INTERFACE I_Reflection

{attribute 'OPC.UA.DA.Property' := '1'}
{attribute 'monitoring' := 'call'}
PROPERTY PUBLIC P_Class : STRING(255)
GET
END_GET
END_PROPERTY

{attribute 'OPC.UA.DA.Property' := '1'}
{attribute 'monitoring' := 'call'}
PROPERTY PUBLIC P_Comment : STRING(255)
GET
END_GET
END_PROPERTY

{attribute 'OPC.UA.DA.Property' := '1'}
{attribute 'monitoring' := 'call'}
PROPERTY PUBLIC P_ID : STRING(25)
GET
END_GET
SET
END_SET
END_PROPERTY

{attribute 'OPC.UA.DA.Property' := '1'}
{attribute 'monitoring' := 'call'}
PROPERTY PUBLIC P_Instance : STRING(255)
GET
END_GET
END_PROPERTY

{attribute 'OPC.UA.DA.Property' := '1'}
{attribute 'monitoring' := 'call'}
PROPERTY PUBLIC P_Timestamp : DT
GET
END_GET
END_PROPERTY

END_INTERFACE

(* stored: Version 1.1.0.1
   Itf I_Reflection: Id {62aeab96-2429-49a4-b102-a608a3391a9f}
   Property P_Class: Id {cbc4d901-48b2-4e97-9d77-884fb0854f2f}
   Get Get: Id {9ab4d9fd-c087-473a-be35-5661f24836f2}
   Property P_Comment: Id {f8cad2c1-c823-4908-b22c-bf669c46c6ef}
   Get Get: Id {83892f6a-bbdf-4950-9818-7b29a5f63cc7}
   Property P_ID: Id {1189c098-5eec-0d68-18e7-7614f6e3884e}
   Get Get: Id {119ce5e0-3bc0-09ab-2641-05ccee762aba}
   Set Set: Id {681c1b60-d8b1-03de-1397-a3678979d92b}
   Property P_Instance: Id {30879d95-d4f4-4455-aa95-646545220952}
   Get Get: Id {e37e3208-271a-4637-87e5-41b8db5cfa3f}
   Property P_Timestamp: Id {d32c7dd1-ae0e-4b1a-b50b-ce8720cabd0c}
   Get Get: Id {e41a45ff-6cea-4e2b-8499-2e70f12a2058} *)
